FUNCTION_BLOCK FB_SuctionCup IMPLEMENTS I_SuctionCup
VAR_INPUT
END_VAR
VAR_OUTPUT
END_VAR
VAR
	fPressure 		AT %I*	: REAL;
	bSuck			AT %Q*	: BOOL;
	bPressure		AT %I* 	: BOOL;
END_VAR

PROPERTY bIsSuck : BOOL
GET
bIsSuck := bPressure;
END_GET
END_PROPERTY

PROPERTY fThreshold : REAL
GET
fThreshold := 6;
END_GET
SET
END_SET
END_PROPERTY

METHOD Release : BOOL
VAR_INPUT
END_VAR
bSuck := FALSE;
END_METHOD

METHOD Suck : BOOL
VAR_INPUT
END_VAR
bSuck := TRUE;
END_METHOD

END_FUNCTION_BLOCK

(* stored: Version 1.1.0.1, ProductVersion 3.1.4024.12
   POU FB_SuctionCup: Id {d16da08f-69a9-440f-8644-b99114ab9a9c}, SpecialFunc None
   Property bIsSuck: Id {31a28ef6-e844-47fe-9440-2b6e84e94a32}
   Get Get: Id {2a39f54a-0e74-4bf5-8dd0-d05b1ba3f090}
   Property fThreshold: Id {e3addf55-7b71-4c3a-8199-ebd63c9ae2f3}
   Get Get: Id {3c7a6992-3317-4c18-ab65-6dd104ad0c44}
   Set Set: Id {88495eee-039f-43df-9a0d-07b42801ea5f}
   Method Release: Id {9c9ac9c3-f3c6-4efe-b31f-2ed47b802dae}
   Method Suck: Id {592836a1-69b9-45a3-b1f4-75215dffbfc3} *)
